{attribute 'qualified_only'}
{attribute 'strict'}
{attribute 'to_string'}
TYPE EN_RobotMessaging :
(
	clearedCmd 					:=10000,
	ok							:=10001,
	retry						:=10002,
	skip						:=10003,
	retriesExceeded				:=10004,
	
	initStart					:=0,
	waitInitPermissive			:=10,
	turnMotorsOFF				:=20,
	waitRobotInAuto				:=30,
	resetEStop					:=40,
	PPToMain					:=50,
	turnMotorsON				:=60,
	startTaskExecuion			:=70,
	waitInitFinihsed			:=80,
	waitRetrievalPerm			:=210,
	stopTaskExecution			:=310,
	initEndMotorsOFF			:=320,
	initFinished				:=999,
	
	autoStarts					,
	waitingPickPerm				,
	pickingGood					,
	pickingNG					,
	waitingPieceStatus			,
	waitingPlacePerm			,
	placing						,
	placeFinished				,
	waitingRejectPerm			,
	rejecting					,
	rejectFinished				,
	autoCycleFinished			:=1999,
	
	manualRetrieval				,
	manualHomming				,
	manualPick					,
	manualCycPickTeach			,
	manualPlace					,
	manualCycPlaceTeach			,
	manualReject				,
	manualCycRejectTeach		
)DINT := clearedCmd;
END_TYPE

(* stored: Version 1.1.0.1, ProductVersion 3.1.4024.12
   DUT EN_RobotMessaging: Id {b82cd2ff-aedf-4a46-a332-f9752b39847d} *)
